# EPICS autosave request: apps/myaDataApp/Db/logEntryData.req
$(P)$(R)logNumber
$(P)$(R)logURL
